PROGRAM MAIN
VAR
	EtherCATIOFactory : EtherCATFactory;
	GetEtherCATDevice: BOOL;
	myDevcie : I_EtherCATDevice;
	CheckMyDevice: BOOL;
	value: BOOL;
END_VAR

IF GetEtherCATDevice THEN
	GetEtherCATDevice := FALSE;
	myDevcie := EtherCATIOFactory.CreateEtherCATDevice();
END_IF

IF CheckMyDevice THEN
	CheckMyDevice := false;
    value := myDevcie.IsDeviceOK();
END_IF

END_PROGRAM

(* stored: Version 1.1.0.1, ProductVersion 3.1.4024.12
   POU MAIN: Id {f4d981b9-50f1-49ec-a1bc-185ecdd2e921}, SpecialFunc None *)
